(* IEC 61131-3 sources: AXOpen/src/components.rexroth.drives/ctrl/test, 2 files *)

(* ---- AxoIndraDriveTests.st ---- *)
// USING AXOpen.Components.Example;
USING AXOpen.Core;
USING AXOpen.Rtc;
USING AXOpen.Logging;

NAMESPACE AxoIndraDriveTests.Tests
    {S7.extern=ReadWrite}
    CLASS TestContext IMPLEMENTS AXOpen.Core.IAxoContext
        VAR
            _openCounter : ULINT;
            _closeCounter : ULINT;
        END_VAR

        METHOD PUBLIC Open : ULINT
            _openCounter := _openCounter + ULINT#1;
        END_METHOD

        METHOD PUBLIC Close : ULINT
            _closeCounter := _closeCounter + ULINT#1;
        END_METHOD

        METHOD PUBLIC CreateIdentity : ULINT
            ;
        END_METHOD

        METHOD PUBLIC OpenCycleCount : ULINT
            OpenCycleCount := _openCounter;
        END_METHOD

        METHOD PUBLIC GetRtc : AXOpen.Rtc.IAxoRtc
            ;
        END_METHOD

        METHOD PUBLIC InjectRtc
            VAR_INPUT
                Rtc : IAxoRtc;
            END_VAR

            ;
        END_METHOD

        METHOD PUBLIC GetLogger : IAxoLogger
            ;
        END_METHOD

        METHOD PUBLIC InjectLogger
            VAR_INPUT
                _logger : IAxoLogger;
            END_VAR

            ;
        END_METHOD
    END_CLASS
    {TestFixture}
    {S7.extern=ReadWrite}
    CLASS AxoIndraDriveTests
        VAR
            context : TestContext;
            drive   : AXOpen.Components.Rexroth.Drives.AxoIndraDrive;
            _AxisIn          :   ARRAY[0..10] OF BYTE;       //  Input data of the axis
            _AxisOut         :   ARRAY[0..10] OF BYTE;       //  Output data of the axis
            _Enable          :   BOOL;                       //  As long as ‘Enable’ is true, power is being enabled.
            _EnablePositive  :   BOOL;                       //  As long as ‘Enable’ is true, this permits motion in positive direction
            _EnableNegative  :   BOOL;                       //  As long as ‘Enable’ is true, this permits motion in negative direction
            _busy : BOOL;
        END_VAR
        {Test}
        METHOD PUBLIC AxoHome
            AxUnit.Assert.Equal(TRUE,TRUE);
        END_METHOD
    END_CLASS
END_NAMESPACE

(* ---- AxoRexrothDriveTests.st ---- *)
USING AXOpen.Components.Rexroth.Drives;
USING AXOpen.Core;
USING AXOpen.Rtc;
USING AXOpen.Logging;

NAMESPACE AxoRexrothDrive.Tests
    CLASS TestContext IMPLEMENTS AXOpen.Core.IAxoContext
        VAR
            _openCounter : ULINT;
            _closeCounter : ULINT;
        END_VAR

        METHOD PUBLIC Open : ULINT
            _openCounter := _openCounter + ULINT#1;
        END_METHOD

        METHOD PUBLIC Close : ULINT
            _closeCounter := _closeCounter + ULINT#1;
        END_METHOD

        METHOD PUBLIC CreateIdentity : ULINT
            ;
        END_METHOD

        METHOD PUBLIC OpenCycleCount : ULINT
            OpenCycleCount := _openCounter;
        END_METHOD

        METHOD PUBLIC GetRtc : AXOpen.Rtc.IAxoRtc
            ;
        END_METHOD

        METHOD PUBLIC InjectRtc
            VAR_INPUT
                Rtc : IAxoRtc;
            END_VAR

            ;
        END_METHOD

        METHOD PUBLIC GetLogger : IAxoLogger
            ;
        END_METHOD

        METHOD PUBLIC InjectLogger
            VAR_INPUT
                _logger : IAxoLogger;
            END_VAR

            ;
        END_METHOD
    END_CLASS
    {TestFixture}
    CLASS CylinderTests
        VAR
            context : TestContext;
            drive : AxoIndraDrive;
            _refAxisIn       :   REF_TO  ARRAY[*] OF BYTE;   //  Reference to the input data of the axis
            _refAxisOut      :   REF_TO  ARRAY[*] OF BYTE;   //  Reference to the output data of the axis

            _done : BOOL;
        END_VAR
        {Test}
        METHOD PUBLIC AxoReset
            WHILE _done DO
                context.Open();
                drive.AxoReset();
                drive.Run(context, _refAxisIn, _refAxisOut, FALSE, FALSE, FALSE);
                AxUnit.Assert.Equal(FALSE, FALSE);
                context.Close();
            END_WHILE;

        END_METHOD
    END_CLASS
END_NAMESPACE
